Yaskawa INFORM job: NULL.JBI

/JOB
//NAME NULL
//POS
///NPOS 0,0,0,0
//INST
///DATE 2014/11/07 21:26
///ATTR 0,0,0,0,0,0,0,0,0,0,0,0,0,0,0,0
///FRAME BASE
NOP
END
